# EPICS StreamDevice protocol: iocTops/VarianTurboPump/VarianTurboPumpApp/Db/tmp/Varian_TPS.proto
ExtraInput = Ignore;
STX = \02;
ADDR = \x80;
ACK = \06;
ETX = \03;
ReplyTimeout = 500;

#
# These are protocols common to all models.
#

getStart {
  out "\${STX}\${ADDR}0000\${ETX}%01<xor8>";
  in  "\${STX}\${ADDR}000%d\${ETX}%01<xor8>";
}

setStart {
  out "\${STX}\${ADDR}0001%{0|1}\${ETX}%01<xor8>";
  in  "\${STX}\${ADDR}\${ACK}\${ETX}%01<xor8>";
  @init { getStart;}
}

getBaudRate {
  out "\${STX}\${ADDR}1080\${ETX}%01<xor8>";
  in  "\${STX}\${ADDR}108%d\${ETX}%01<xor8>";
}

setBaudRate {
  out "\${STX}\${ADDR}1081%06d\${ETX}%01<xor8>";
  in  "\${STX}\${ADDR}\${ACK}\${ETX}%01<xor8>";
  @init { getBaudRate;}
}

getCurrent {
  out "\${STX}\${ADDR}2000\${ETX}%01<xor8>";
  in  "\${STX}\${ADDR}200%f\${ETX}%01<xor8>";
}

getVoltage {
  out "\${STX}\${ADDR}2010\${ETX}%01<xor8>";
  in  "\${STX}\${ADDR}201%f\${ETX}%01<xor8>";
}

getErrorCode {
  out "\${STX}\${ADDR}2060\${ETX}%01<xor8>";
  in  "\${STX}\${ADDR}206%d\${ETX}%01<xor8>";
}

#
# This traps error responses
# Be sure to set SCAN field to "I/O Intr"
#
trapErrors {
  in  "\${STX}\${ADDR}%{\xff|\x15|\x32|\x33|\x34|\x35}\${ETX}%01<xor8>";
}
#
# These are protocols specific to the Varian TPS-compact
#

getLowSpeed {
  out "\${STX}\${ADDR}0010\${ETX}%01<xor8>";
  in  "\${STX}\${ADDR}001%d\${ETX}%01<xor8>";
}

setLowSpeed {
  out "\${STX}\${ADDR}0011%{0|1}\${ETX}%01<xor8>";
  in  "\${STX}\${ADDR}\${ACK}\${ETX}%01<xor8>";
  @init { getLowSpeed;}
}

getCtrlMode {
  out "\${STX}\${ADDR}0080\${ETX}%01<xor8>";
  in  "\${STX}\${ADDR}008%d\${ETX}%01<xor8>";
}

setCtrlMode {
  out "\${STX}\${ADDR}0081%{0|1}\${ETX}%01<xor8>";
  in  "\${STX}\${ADDR}\${ACK}\${ETX}%01<xor8>";
  @init { getCtrlMode;}
}

getSoftStart {
  out "\${STX}\${ADDR}1000\${ETX}%01<xor8>";
  in  "\${STX}\${ADDR}100%d\${ETX}%01<xor8>";
}

setSoftStart {
  out "\${STX}\${ADDR}1001%{0|1}\${ETX}%01<xor8>";
  in  "\${STX}\${ADDR}\${ACK}\${ETX}%01<xor8>";
  @init { getSoftStart;}
}

getSP1Type {
  out "\${STX}\${ADDR}1010\${ETX}%01<xor8>";
  in  "\${STX}\${ADDR}101%d\${ETX}%01<xor8>";
}

setSP1Type {
  out "\${STX}\${ADDR}1011%06d\${ETX}%01<xor8>";
  in  "\${STX}\${ADDR}\${ACK}\${ETX}%01<xor8>";
  @init { getSP1Type;}
}

getSetPoint {
  out "\${STX}\${ADDR}1020\${ETX}%01<xor8>";
  in  "\${STX}\${ADDR}102%d\${ETX}%01<xor8>";
}

setSetPoint {
  out "\${STX}\${ADDR}1021%06d\${ETX}%01<xor8>";
  in  "\${STX}\${ADDR}\${ACK}\${ETX}%01<xor8>";
  @init { getSetPoint;}
}

getSP1Delay {
  out "\${STX}\${ADDR}1030\${ETX}%01<xor8>";
  in  "\${STX}\${ADDR}103%d\${ETX}%01<xor8>";
}

setSP1Delay {
  out "\${STX}\${ADDR}1031%06d\${ETX}%01<xor8>";
  in  "\${STX}\${ADDR}\${ACK}\${ETX}%01<xor8>";
  @init { getSP1Delay;}
}

getSP1Signal {
  out "\${STX}\${ADDR}1040\${ETX}%01<xor8>";
  in  "\${STX}\${ADDR}104%d\${ETX}%01<xor8>";
}

setSP1Signal {
  out "\${STX}\${ADDR}1041%{0|1}\${ETX}%01<xor8>";
  in  "\${STX}\${ADDR}\${ACK}\${ETX}%01<xor8>";
  @init { getSP1Signal;}
}

getSP1Hyst {
  out "\${STX}\${ADDR}1050\${ETX}%01<xor8>";
  in  "\${STX}\${ADDR}105%d\${ETX}%01<xor8>";
}

setSP1Hyst {
  out "\${STX}\${ADDR}1051%06d\${ETX}%01<xor8>";
  in  "\${STX}\${ADDR}\${ACK}\${ETX}%01<xor8>";
  @init { getSP1Hyst;}
}

getWaterCooled {
  out "\${STX}\${ADDR}1060\${ETX}%01<xor8>";
  in  "\${STX}\${ADDR}106%d\${ETX}%01<xor8>";
}

setWaterCooled {
  out "\${STX}\${ADDR}1061%{0|1}\${ETX}%01<xor8>";
  in  "\${STX}\${ADDR}\${ACK}\${ETX}%01<xor8>";
  @init { getWaterCooled;}
}

getActiveStop {
  out "\${STX}\${ADDR}1070\${ETX}%01<xor8>";
  in  "\${STX}\${ADDR}107%d\${ETX}%01<xor8>";
}

setActiveStop {
  out "\${STX}\${ADDR}1071%{0|1}\${ETX}%01<xor8>";
  in  "\${STX}\${ADDR}\${ACK}\${ETX}%01<xor8>";
  @init { getActiveStop;}
}

setResetCounters {
  out "\${STX}\${ADDR}1091%{0|1}\${ETX}%01<xor8>";
  in  "\${STX}\${ADDR}\${ACK}\${ETX}%01<xor8>";
}

getInterlockType {
  out "\${STX}\${ADDR}1100\${ETX}%01<xor8>";
  in  "\${STX}\${ADDR}110%d\${ETX}%01<xor8>";
}

setInterlockType {
  out "\${STX}\${ADDR}1101%{0|1}\${ETX}%01<xor8>";
  in  "\${STX}\${ADDR}\${ACK}\${ETX}%01<xor8>";
  @init { getInterlockType;}
}

getAnalogOutType {
  out "\${STX}\${ADDR}1110\${ETX}%01<xor8>";
  in  "\${STX}\${ADDR}111%d\${ETX}%01<xor8>";
}

setAnalogOutType {
  out "\${STX}\${ADDR}1111%06d\${ETX}%01<xor8>";
  in  "\${STX}\${ADDR}\${ACK}\${ETX}%01<xor8>";
  @init { getAnalogOutType;}
}

getLowSpeedFreq {
  out "\${STX}\${ADDR}1170\${ETX}%01<xor8>";
  in  "\${STX}\${ADDR}117%d\${ETX}%01<xor8>";
}

setLowSpeedFreq {
  out "\${STX}\${ADDR}1171%06d\${ETX}%01<xor8>";
  in  "\${STX}\${ADDR}\${ACK}\${ETX}%01<xor8>";
  @init { getLowSpeedFreq;}
}

getRotFreq {
  out "\${STX}\${ADDR}1200\${ETX}%01<xor8>";
  in  "\${STX}\${ADDR}120%d\${ETX}%01<xor8>";
}

setRotFreq {
  out "\${STX}\${ADDR}1201%06d\${ETX}%01<xor8>";
  in  "\${STX}\${ADDR}\${ACK}\${ETX}%01<xor8>";
  @init { getRotFreq;}
}

getMaxRotFreq {
  # code 121 not supported
  wait 0;
}

setMaxRotFreq {
  # code 121 not supported
  wait 0;
}

getVentValve {
  out "\${STX}\${ADDR}1220\${ETX}%01<xor8>";
  in  "\${STX}\${ADDR}122%d\${ETX}%01<xor8>";
}

setVentValve {
  out "\${STX}\${ADDR}1221%{0|1}\${ETX}%01<xor8>";
  in  "\${STX}\${ADDR}\${ACK}\${ETX}%01<xor8>";
  @init { getVentValve;}
}

getVentValveMode {
  out "\${STX}\${ADDR}1250\${ETX}%01<xor8>";
  in  "\${STX}\${ADDR}125%d\${ETX}%01<xor8>";
}

setVentValveMode {
  out "\${STX}\${ADDR}1251%{0|1}\${ETX}%01<xor8>";
  in  "\${STX}\${ADDR}\${ACK}\${ETX}%01<xor8>";
  @init { getVentValveMode;}
}

getVentValveDelay {
  out "\${STX}\${ADDR}1260\${ETX}%01<xor8>";
  in  "\${STX}\${ADDR}126%d\${ETX}%01<xor8>";
}

setVentValveDelay {
  out "\${STX}\${ADDR}1261%06d\${ETX}%01<xor8>";
  in  "\${STX}\${ADDR}\${ACK}\${ETX}%01<xor8>";
  @init { getVentValveDelay;}
}

getGaugeSPType {
  # code 136 not supported
  wait 0;
}

setGaugeSPType {
  # code 136 not supported
  wait 0;
}

getGaugeSP {
  # code 137 not supported
  wait 0;
}

setGaugeSP {
  # code 137 not supported
  wait 0;
}

getGaugeSPDelay {
  # code 138 not supported
  wait 0;
}

setGaugeSPDelay {
  # code 138 not supported
  wait 0;
}

getGaugeSPSignal {
  # code 139 not supported
  wait 0;
}

setGaugeSPSignal {
  # code 139 not supported
  wait 0;
}

getGaugeSPHyst {
  # code 140 not supported
  wait 0;
}

setGaugeSPHyst {
  # code 140 not supported
  wait 0;
}

getExtFanConfig {
  # code 143 not supported
  wait 0;
}

setExtFanConfig {
  # code 143 not supported
  wait 0;
}

getExtFan {
  # code 144 not supported
  wait 0;
}

setExtFan {
  # code 144 not supported
  wait 0;
}

getVentOpenTime {
  out "\${STX}\${ADDR}1470\${ETX}%01<xor8>";
  in  "\${STX}\${ADDR}147%d\${ETX}%01<xor8>";
}

setVentOpenTime {
  out "\${STX}\${ADDR}1471%06d\${ETX}%01<xor8>";
  in  "\${STX}\${ADDR}\${ACK}\${ETX}%01<xor8>";
  @init { getVentOpenTime;}
}

getPowerLimit {
  out "\${STX}\${ADDR}1550\${ETX}%01<xor8>";
  in  "\${STX}\${ADDR}155%d\${ETX}%01<xor8>";
}

getLoadtype {
  out "\${STX}\${ADDR}1570\${ETX}%01<xor8>";
  in  "\${STX}\${ADDR}157%d\${ETX}%01<xor8>";
}

setLoadtype {
  out "\${STX}\${ADDR}1571%06d\${ETX}%01<xor8>";
  in  "\${STX}\${ADDR}\${ACK}\${ETX}%01<xor8>";
  @init { getLoadtype;}
}

getGaugePCorr {
  out "\${STX}\${ADDR}1610\${ETX}%01<xor8>";
  in  "\${STX}\${ADDR}161%d\${ETX}%01<xor8>";
}

setGaugePCorr {
  out "\${STX}\${ADDR}1611%06d\${ETX}%01<xor8>";
  in  "\${STX}\${ADDR}\${ACK}\${ETX}%01<xor8>";
  @init { getGaugePCorr;}
}

# there is white space between the data and ETX and the
# protocol parser does not ignore it
getSP1Press {
  out "\${STX}\${ADDR}1620\${ETX}%01<xor8>";
  in  "\${STX}\${ADDR}162%E%*[ ]\${ETX}%01<xor8>";
}

setSP1Press {
  out "\${STX}\${ADDR}1621%2.1E\${ETX}%01<xor8>";
  in  "\${STX}\${ADDR}\${ACK}\${ETX}%01<xor8>";
  @init { getSP1Press;}
}

getPressUnits {
  out "\${STX}\${ADDR}1630\${ETX}%01<xor8>";
  in  "\${STX}\${ADDR}163%d\${ETX}%01<xor8>";
}

setPressUnits {
  out "\${STX}\${ADDR}1631%06d\${ETX}%01<xor8>";
  in  "\${STX}\${ADDR}\${ACK}\${ETX}%01<xor8>";
  @init { getPressUnits;}
}

getStopSpeedRead {
  out "\${STX}\${ADDR}1670\${ETX}%01<xor8>";
  in  "\${STX}\${ADDR}167%d\${ETX}%01<xor8>";
}

setStopSpeedRead {
  out "\${STX}\${ADDR}1671%10s\${ETX}%01<xor8>";
  in  "\${STX}\${ADDR}\${ACK}\${ETX}%01<xor8>";
  @init { getStopSpeedRead;}
}

getSP2Type {
  # code 171 not supported
  wait 0;
}

setSP2Type {
  # code 171 not supported
  wait 0;
}

getSetPoint2 {
  # code 172 not supported
  wait 0;
}

setSetPoint2 {
  # code 172 not supported
  wait 0;
}

getSP2Delay {
  # code 173 not supported
  wait 0;
}

setSP2Delay {
  # code 173 not supported
  wait 0;
}

getSP2Signal {
  # code 174 not supported
  wait 0;
}

setSP2Signal {
  # code 174 not supported
  wait 0;
}

getSP2Hyst {
  # code 175 not supported
  wait 0;
}

setSP2Hyst {
  # code 175 not supported
  wait 0;
}

getSP2Press {
  # code 176 not supported
  wait 0;
}

setSP2Press {
  # code 176 not supported
  wait 0;
}

getStartOutMode {
  # code 177 not supported
  wait 0;
}

setStartOutMode {
  # code 177 not supported
  wait 0;
}

getGasType {
  # code 181 not supported
  wait 0;
}

setGasType {
  # code 181 not supported
  wait 0;
}

getOtherGCorr {
  # code 182 not supported
  wait 0;
}

setOtherGCorr {
  # code 182 not supported
  wait 0;
}

getPower {
  # code 202 not supported
  wait 0;
}

getDrivingFreq {
  # code 203 not supported
  wait 0;
}

getTemperature {
  # code 204 not supported
  wait 0;
}

getStatus {
  # code 205 not supported
  wait 0;
}

getSP1State {
  # code 207 not supported
  wait 0;
}

getSP2State {
  # code 208 not supported
  wait 0;
}

getHeatSinkTemp {
  # code 211 not supported
  wait 0;
}

getAirTemp {
  out "\${STX}\${ADDR}2160\${ETX}%01<xor8>";
  in  "\${STX}\${ADDR}216%f\${ETX}%01<xor8>";
}

getSP1StateA {
  # code 221 not supported
  wait 0;
}

# there is white space between the data and ETX and the
# protocol parser does not ignore it
getPressure{
  out "\${STX}\${ADDR}2240\${ETX}%01<xor8>";
  in  "\${STX}\${ADDR}224%E%*[ ]\${ETX}%01<xor8>";
}

getSP2StateA {
  # code 225 not supported
  wait 0;
}

getFreq {
  out "\${STX}\${ADDR}2260\${ETX}%01<xor8>";
  in  "\${STX}\${ADDR}226%f\${ETX}%01<xor8>";
}

getGaugeStatus {
  # code 257 not supported
  wait 0;
}

getGaugePower {
  # code 267 not supported
  wait 0;
}

setGaugePower {
  # code 267 not supported
  wait 0;
}

getCycleTime {
  out "\${STX}\${ADDR}3000\${ETX}%01<xor8>";
  in  "\${STX}\${ADDR}300%d\${ETX}%01<xor8>";
}

getCycleNumber {
  out "\${STX}\${ADDR}3010\${ETX}%01<xor8>";
  in  "\${STX}\${ADDR}301%d\${ETX}%01<xor8>";
}

getLife {
  out "\${STX}\${ADDR}3020\${ETX}%01<xor8>";
  in  "\${STX}\${ADDR}302%d\${ETX}%01<xor8>";
}

getTipSealLife {
  # code 358 not supported
  wait 0;
}

# there is white space between the data and ETX and the
# protocol parser does not ignore it
getCRCEPROM {
  out "\${STX}\${ADDR}4000\${ETX}%01<xor8>";
  in  "\${STX}\${ADDR}400%s%*[ ]\${ETX}%01<xor8>";
}

getBootCRC {
  # code 401 not supported
  wait 0;
}

# there is white space between the data and ETX and the
# protocol parser does not ignore it
getCRCPar {
  out "\${STX}\${ADDR}4020\${ETX}%01<xor8>";
  in  "\${STX}\${ADDR}402%s%*[ ]\${ETX}%01<xor8>";
}

# there is white space between the data and ETX and the
# protocol parser does not ignore it
getCRCParStruct {
  out "\${STX}\${ADDR}4040\${ETX}%01<xor8>";
  in  "\${STX}\${ADDR}404%s%*[ ]\${ETX}%01<xor8>";
}

# there is white space between the data and ETX and the
# protocol parser does not ignore it
getProgListCode {
  out "\${STX}\${ADDR}4060\${ETX}%01<xor8>";
  in  "\${STX}\${ADDR}406%s%*[ ]\${ETX}%01<xor8>";
}

# there is white space between the data and ETX and the
# protocol parser does not ignore it
getParListCode {
  out "\${STX}\${ADDR}4070\${ETX}%01<xor8>";
  in  "\${STX}\${ADDR}407%s%*[ ]\${ETX}%01<xor8>";
}

getFirmwareRev {
  # code 408 not supported
  wait 0;
}

getSerialAddr {
  out "\${STX}\${ADDR}5030\${ETX}%01<xor8>";
  in  "\${STX}\${ADDR}503%d\${ETX}%01<xor8>";
}

setSerialAddr {
  out "\${STX}\${ADDR}5031%06d\${ETX}%01<xor8>";
  in  "\${STX}\${ADDR}\${ACK}\${ETX}%01<xor8>";
  @init { getSerialAddr;}
}

getSerialType {
  out "\${STX}\${ADDR}5040\${ETX}%01<xor8>";
  in  "\${STX}\${ADDR}504%d\${ETX}%01<xor8>";
}

setSerialType {
  out "\${STX}\${ADDR}5041%{0|1}\${ETX}%01<xor8>";
  in  "\${STX}\${ADDR}\${ACK}\${ETX}%01<xor8>";
  @init { getSerialType;}
}
